tonClickTimer(PT:=tDoubleClickTime);
tonHoldTimer(PT:=tHoldTime);
cClickCnt(CU:=bButton, PV:=2);

// 点击检测
IF bButton AND cClickCnt.CV=1 THEN
	nStep := 1;												// 检测到单击
ELSIF bButton AND cClickCnt.CV=2 THEN
	nStep := 2;												// 检测到双击，进入双击+HOLD模式检测
END_IF



IF tonClickTimer.Q AND NOT bButton THEN						// 第一次单击后开启tonClickTimer计时器，计时器触发且没有检测到按钮按下，则将按键计数器复位，并将状态nstep=0，恢复到默认无按键按下状态。
	cClickCnt(RESET:= TRUE);
	nStep	:= 0;
ELSIF tonClickTimer.Q AND bButton AND cClickCnt.CV=1 THEN	// 第一次单击后开启tonClickTimer计时器，计时器触发且检测到按钮一直被按下。
	nStep := 3;												// 进入单击+HOLD模式
END_IF

// 按键计数器自复位
IF cClickCnt.Q THEN
	cClickCnt(reset:=TRUE);
END_IF




CASE nStep OF
	// 无按键状态，所有定时器计数器复位，两个输出变量bDoubleClickAndHold、bOnceClickAndHold置false
	0:
		tonClickTimer(IN := FALSE);
		tonHoldTimer(IN:=FALSE);
		cClickCnt(RESET:= FALSE);
		bDoubleClickAndHold := FALSE;
		bOnceClickAndHold:=FALSE;
	
	//点击模式检测
	1:
		tonClickTimer(IN:=TRUE);
		
	// 双击+hold检测
	2:
		tonHoldTimer(IN:=TRUE);								//开启hold时间计时器
		
		IF tonHoldTimer.Q AND bButton THEN					// 如果Hold时间满足，即为双击+hold状态
			bDoubleClickAndHold := TRUE;
		END_IF
		
		IF NOT bButton THEN									// 检测到按键释放，所有计时器计数器、输出状态复位
			bDoubleClickAndHold := FALSE;
			tonClickTimer(IN:=FALSE);
			tonHoldTimer(IN:=FALSE);
			cClickCnt(RESET:= TRUE);
			nStep:=0;
		END_IF
	
	// 单击+HOLD模式	
	3:
		IF tonClickTimer.Q AND bButton THEN					// 单击的hold时根据tonClickTimer时间来测量的，时间满足且按键未松，则为单击+hold
			bOnceClickAndHold := TRUE;
		END_IF
		
		IF NOT bButton THEN									// 检测到按键释放，所有计时器计数器、输出状态复位
			bOnceClickAndHold := FALSE;
			tonClickTimer(IN:=FALSE);
			cClickCnt(RESET:= TRUE);
			nStep:=0;
		END_IF
		
END_CASE

END_FUNCTION_BLOCK

// ---- POUs/TBoxCtrl.TcPOU
PROGRAM TBoxCtrl
VAR
END_VAR

IF bPumpMotor_Enable_TBox OR bPumpMotor_Enable_UpperUI THEN
	bPumpMotor_Enable:=TRUE;
ELSE
	bPumpMotor_Enable:=FALSE;
END_IF
	
IF bLeftArm_SV1_TBox OR bLeftArm_SV1_UpperUI THEN
	bLeftArm_SV1:=TRUE;
ELSE
	bLeftArm_SV1:=FALSE;
END_IF

IF bLeftArm_SV2_TBox OR bLeftArm_SV2_UpperUI THEN
	bLeftArm_SV2:=TRUE;
ELSE
	bLeftArm_SV2:=FALSE;
END_IF

IF bLeftArm_SV3_TBox OR bLeftArm_SV3_UpperUI THEN
	bLeftArm_SV3:=TRUE;
ELSE
	bLeftArm_SV3:=FALSE;
END_IF

IF bLeftArm_SV4_TBox OR bLeftArm_SV4_UpperUI THEN
	bLeftArm_SV4:=TRUE;
ELSE
	bLeftArm_SV4:=FALSE;
END_IF

IF bLeftArm_SV5_TBox OR bLeftArm_SV5_UpperUI THEN
	bLeftArm_SV5:=TRUE;
ELSE
	bLeftArm_SV5:=FALSE;
END_IF

IF bLeftArm_SV6_TBox OR bLeftArm_SV6_UpperUI THEN
	bLeftArm_SV6:=TRUE;
ELSE
	bLeftArm_SV6:=FALSE;
END_IF

IF bLeftArm_SV7_TBox OR bLeftArm_SV7_UpperUI THEN
	bLeftArm_SV7:=TRUE;
ELSE
	bLeftArm_SV7:=FALSE;
END_IF

IF bLeftArm_SV8_TBox OR bLeftArm_SV8_UpperUI THEN
	bLeftArm_SV8:=TRUE;
ELSE
	bLeftArm_SV8:=FALSE;
END_IF




IF bRightArm_SV1_TBox OR bRightArm_SV1_UpperUI THEN
	bRightArm_SV1:=TRUE;
ELSE
	bRightArm_SV1:=FALSE;
END_IF

IF bRightArm_SV2_TBox OR bRightArm_SV2_UpperUI THEN
	bRightArm_SV2:=TRUE;
ELSE
	bRightArm_SV2:=FALSE;
END_IF

IF bRightArm_SV3_TBox OR bRightArm_SV3_UpperUI THEN
	bRightArm_SV3:=TRUE;
ELSE
	bRightArm_SV3:=FALSE;
END_IF

IF bRightArm_SV4_TBox OR bRightArm_SV4_UpperUI THEN
	bRightArm_SV4:=TRUE;
ELSE
	bRightArm_SV4:=FALSE;
END_IF

IF bRightArm_SV5_TBox OR bRightArm_SV5_UpperUI THEN
	bRightArm_SV5:=TRUE;
ELSE
	bRightArm_SV5:=FALSE;
END_IF

IF bRightArm_SV6_TBox OR bRightArm_SV6_UpperUI THEN
	bRightArm_SV6:=TRUE;
ELSE
	bRightArm_SV6:=FALSE;
END_IF

IF bRightArm_SV7_TBox OR bRightArm_SV7_UpperUI THEN
	bRightArm_SV7:=TRUE;
ELSE
	bRightArm_SV7:=FALSE;
END_IF

IF bRightArm_SV8_TBox OR bRightArm_SV8_UpperUI THEN
	bRightArm_SV8:=TRUE;
ELSE
	bRightArm_SV8:=FALSE;
END_IF

END_PROGRAM

// ---- POUs/AxisStatus.TcPOU
PROGRAM AxisStatus
VAR
	


RE:AxisStatusReadErrorCode;





END_VAR

axis_RightArm_Left();
axis_RightArm_Right();
axis_RightArm_Wrist();
axis_RightArm_Lift();
axis_LeftArm_Left();
axis_LeftArm_Right();
axis_LeftArm_Wrist();
axis_LeftArm_Lift();
axis_SmallGate_Left();
axis_SmallGate_Right();
axis_BigGate_Left();
axis_BigGate_Right();
axis_BackGate_Left();
axis_BackGate_Right();

END_PROGRAM

// ---- POUs/AxisStatusReadErrorCode.TcPOU
FUNCTION_BLOCK AxisStatusReadErrorCode
VAR_INPUT
	AxisName				:AXIS_REF;

END_VAR
VAR_OUTPUT
	ErrorCode				:STRING;
	nMainAlarmCode			: USINT;
	nSubAlarmCode			: USINT;
END_VAR
VAR
	fbReadDriverSDO			: FB_EcCoeSdoRead;
	receivedAlarmCode		: UDINT;
//	nMainAlarmCode			: USINT;
//	nSubAlarmCode			: USINT;
	
	
END_VAR

fbReadDriverSDO(
	sNetId:= '192.168.1.20.1.1', 
	nSlaveAddr:= 1014, 
	nSubIndex:= 16#02, 
	nIndex:= 16#4DA0, 
	pDstBuf:= ADR(receivedAlarmCode), 
	cbBufLen:= 8, 
	bExecute:= , 
	tTimeout:= , 
	bBusy=> , 
	bError=> , 
	nErrId=> , 
	cbRead=> );
	
//0111 1111 1111 1111
//7F		FF
//nMainAlarmCode  := receivedAlarmCode AND SHL(16#0000007F, 8);
//nSubAlarmCode	:= receivedAlarmCode AND SHL(16#000000FF, 0);
nMainAlarmCode := TO_USINT(SHR(receivedAlarmCode, 8)) AND (16#7F);
nSubAlarmCode := TO_USINT(receivedAlarmCode) AND (16#FF);

END_FUNCTION_BLOCK

// ---- POUs/LedControl.TcPOU
PROGRAM LedControl
VAR
	
	
	
	
END_VAR

END_PROGRAM

// ---- POUs/LedLogic.TcPOU
FUNCTION_BLOCK LedLogic
VAR_INPUT
END_VAR
VAR_OUTPUT
END_VAR
VAR
END_VAR

END_FUNCTION_BLOCK

// ---- POUs/ArmFK_bak.TcPOU
FUNCTION ArmFK_bak : Points
VAR_INPUT
	theta1:LREAL;
	theta2:LREAL;
END_VAR
VAR
	// 中间变量
	theta1_rad:LREAL;
	theta2_rad:LREAL;
	rr:LREAL;						//r变量被倍福占用了，所以此处用rr
	u:LREAL;
	angle_ACD:LREAL;
	angle_DCE:LREAL;
	angle_ACF:LREAL;
	angle_FCG:LREAL;
	angle_FCI:LREAL;
	
	// 输出
	points : Points;

END_VAR

(*

theta1_rad := DEG_TO_RAD(theta1);
theta2_rad := DEG_TO_RAD(theta2);


rr := SQRT(EXPT((2*w+f*COS(theta1_rad)-g*COS(theta2_rad)),2) + EXPT((f*SIN(theta1_rad)-g*SIN(theta2_rad)),2));  

u := SQRT(EXPT((2*w-g*COS(theta2_rad)),2) + EXPT((-g*SIN(theta2_rad)),2));


angle_ACD := ACOS((rr*rr+f*f-u*u)/(2*rr*f));


angle_DCE := ACOS((rr*rr + i*i -h*h)/(2*rr*i));


angle_ACF := angle_ACD + angle_DCE + DEG_TO_RAD(angle_FCE);


angle_FCG := angle_ACF - theta1_rad;


angle_FCI := PI - angle_FCG;
points.x := w + f*COS(theta1_rad) + n*COS(angle_FCI);
points.y := f*SIN(theta1_rad) + n*SIN(angle_FCI);

ArmLeftFK := points;

*)

END_FUNCTION

// ---- POUs/ArmIK_bak.TcPOU
FUNCTION ArmIK_bak : Angles
VAR_INPUT
	x:LREAL;
	y:LREAL;
END_VAR
VAR
	
	// 中间量
	p:LREAL;
	q:LREAL;
	l:LREAL;
	k:LREAL;
	angle_CAF:LREAL;	
	angle_OAF:LREAL;
	theta1:LREAL;
	theta2:LREAL;
	angle_ACF:LREAL;
	angle_ACE:LREAL;
	angle_CAE:LREAL;
	angle_EAB:LREAL;
	angle_EBA:LREAL;
	angle_DBE:LREAL;
	
	// 输出
	angles		:Angles;
	
END_VAR

// TWINCAT 角度换算以弧度为单位
(*

p := SQRT((x-w)*(x-w)+y*y);
q := SQRT(x*x + y*y);
 
//n := SQRT(i*i+j*j-2*i*j*COS(DEG_TO_RAD(angle_a)));
angle_CAF := ACOS((f*f+p*p-n*n)/(2*f*p));
angle_OAF := ACOS((w*w+p*p-q*q)/(2*w*p));
theta1 := PI-angle_CAF-angle_OAF;

angle_ACF := ACOS((f*f+n*n-p*p)/(2*f*n));
//angle_FCE := ACOS((n*n+i*i-j*j)/(2*n*i));
angle_ACE := angle_ACF - DEG_TO_RAD(angle_FCE);
l := SQRT(i*i+f*f-2*i*f*COS(angle_ACE));
angle_CAE := ACOS((f*f+l*l-i*i)/(2*f*l));
angle_EAB := PI-theta1 - angle_CAE;
k := SQRT(l*l + 4*w*w - 4*l*w*COS(angle_EAB));
angle_EBA := ACOS((k*k+4*w*w-l*l)/(4*k*w));
angle_DBE := ACOS((g*g+k*k-h*h)/(2*g*k));
theta2 := angle_EBA + angle_DBE;

angles.theta1_right := RAD_TO_DEG(theta1);
angles.theta2_left := RAD_TO_DEG(theta2);


ArmLeftIK := angles;

*)

END_FUNCTION

// ---- POUs/ArmMove.TcPOU
PROGRAM ArmMove
VAR
	
	point												:Points;					// 当前腕关节坐标
	target_angle										:Angles;					// 臂左右电机目标角度
	manualState											:USINT;						// 手动控制状态标志位，0
	speed												:REAL := 1;					// 笛卡尔坐标位移速度
	x													:REAL;						// 腕关节目标位置x
	y													:REAL;						// 腕关节目标位置y
	wrist_angle											:REAL;
	wrist_MoveAbs										:MC_MoveAbsolute;
	
	LeftArm_Right_ExtPosGen_Enable						:MC_ExtSetPointGenEnable;
	LeftArm_Right_ExtPosGen_Disable                     :MC_ExtSetPointGenDisable;
	LeftArm_Left_ExtPosGen_Enable                       :MC_ExtSetPointGenEnable;
	LeftArm_Left_ExtPosGen_Disable	                    :MC_ExtSetPointGenDisable;
	
	fb_SerialCom		:FB_SerialCom;					//串口
	wrist_angle_int		:INT;
	wrist_angle_byte	:BYTE;
	
	
END_VAR

axis_LeftArm_Left();
axis_LeftArm_Right();
ExtPosGen();

// 外部位置发生器失能
LeftArm_Right_ExtPosGen_Enable.Execute 		:= FALSE;
LeftArm_Right_ExtPosGen_Disable.Execute 	:= FALSE;
LeftArm_Left_ExtPosGen_Enable.Execute 		:= FALSE;
LeftArm_Left_ExtPosGen_Disable.Execute 		:= FALSE;

IF bManualCtrl_Part_LeftArm_Left THEN
	
	// 运动学正解出当前腕关节点坐标
	point := ArmFK(axis_LeftArm_Right.NcToPlc.ActPos, axis_LeftArm_Left.NcToPlc.ActPos);
	
	// 用舵机进行程序验证的串口背景通讯
	//BackgroundSerialCtrl();
	
	IF bAutoCtrl_Part_LeftWrist THEN
		
		wrist_angle := WristIK(point.x, point.y);		// 逆解出腕电机角度
		wrist_angle_int:= TO_INT(wrist_angle);
		
		// 用舵机进行程序验证的串口测试
		//wrist_angle_byte:= INT_TO_BYTE(wrist_angle_int);
		//fb_SerialCom(TxBuffer:= TxBuffer, RxBuffer:= RxBuffer, angle:= wrist_angle_byte);	
		
		wrist_MoveAbs(Axis:= axis_LeftArm_Wrist, Execute:= TRUE, Position:= wrist_angle, Velocity:= 5, Acceleration:= 10, Deceleration:= , Jerk:= , BufferMode:= , 
					  Options:= , Done=> , Busy=> , Active=> , CommandAborted=> , Error=> , ErrorID=> );		// 腕电机走绝对定位
	END_IF
	

	IF bLeftArm_Forward THEN
		x := point.x;
		y := point.y + speed;
		target_angle := ArmIK(x, y);
		manualState := 1;
		
	ELSIF bLeftArm_Backward THEN
	
		x := point.x;
		y := point.y - speed;
		target_angle := ArmIK(x, y);
		manualState := 1;
		
	ELSIF bLeftArm_Left THEN
		
		x := point.x - speed;
		y := point.y;
		target_angle := ArmIK(x, y);
		manualState := 1;
		
	ELSIF bLeftArm_Right THEN
		
		x := point.x + speed;
		y := point.y;
		target_angle := ArmIK(x, y);
		manualState := 1;
		
	ELSE
		manualState := 0;
	END_IF
	
	
	
	CASE manualState OF
		0:
			LeftArm_Right_ExtPosGen_Enable.Execute 		:= FALSE;
			LeftArm_Right_ExtPosGen_Disable.Execute 	:= TRUE;
			LeftArm_Left_ExtPosGen_Enable.Execute 		:= FALSE;
			LeftArm_Left_ExtPosGen_Disable.Execute 		:= TRUE;
		
		1:
			LeftArm_Right_ExtPosGen_Enable.Execute := TRUE;
			LeftArm_Left_ExtPosGen_Enable.Execute := TRUE;
			IF axis_LeftArm_Right.Status.ExtSetPointGenEnabled AND axis_LeftArm_Left.Status.ExtSetPointGenEnabled THEN
				MC_ExtSetPointGenFeed(
					Position:= target_angle.theta1_right, 
					Velocity:= 30,  
					Acceleration:= 10,  
					Direction:= 1, 
					Axis:= axis_LeftArm_Right);
		
				MC_ExtSetPointGenFeed(
					Position:= target_angle.theta2_left, 
					Velocity:= 30,  
					Acceleration:= 10,  
					Direction:= 1, 
					Axis:= axis_LeftArm_Left);
			END_IF
	END_CASE

//ELSE

END_IF

ACTION ExtPosGen:
LeftArm_Right_ExtPosGen_Enable(
	Axis:= axis_LeftArm_Right, 
	Execute:= LeftArm_Right_ExtPosGen_Enable.Execute, 
	Position:= , 
	PositionType:= , 
	Done=> , 
	Busy=> , 
	Error=> , 
	ErrorID=> , 
	Enabled=> );
	
LeftArm_Right_ExtPosGen_Disable(
	Axis:= axis_LeftArm_Right, 
	Execute:= LeftArm_Right_ExtPosGen_Disable.Execute, 
	Done=> , 
	Busy=> , 
	Error=> , 
	ErrorID=> , 
	Enabled=> );
	
LeftArm_Left_ExtPosGen_Enable(
	Axis:= axis_LeftArm_Left, 
	Execute:= LeftArm_Left_ExtPosGen_Enable.Execute, 
	Position:= , 
	PositionType:= , 
	Done=> , 
	Busy=> , 
	Error=> , 
	ErrorID=> , 
	Enabled=> );
	
LeftArm_Left_ExtPosGen_Disable(
	Axis:= axis_LeftArm_Left, 
	Execute:= LeftArm_Left_ExtPosGen_Disable.Execute, 
	Done=> , 
	Busy=> , 
	Error=> , 
	ErrorID=> , 
	Enabled=> );
END_ACTION

END_PROGRAM

// ---- POUs/AxisCaliHomePos.TcPOU
PROGRAM AxisCaliHomePos
VAR
	writeParam		:MC_WriteParameter;
	bWriteParam_DO	:BOOL;
	
END_VAR


writeParam(
	Axis:= axis_RightArm_Wrist, 
	Execute:= bWriteParam_DO, 
	ParameterNumber:= AxisEncoderOffset, 
	Value:= -2, 
	Done=> , 
	Busy=> , 
	Error=> , 
	ErrorID=> );

END_PROGRAM

// ---- POUs/Gate_Back_Move.TcPOU
PROGRAM Gate_Back_Move
VAR
	
	backGateGearIn					:MC_GearIn;
	backGateGearOut					:MC_GearOut;	                    			
	backGateLeftAxisJog 			:MC_Jog;
	backGateLeftAxisMoveAbs			:MC_MoveAbsolute;		// 后龙门MoveAbs(实际上电子齿轮的Master轴axis_BackGate_Left的Mc_MoveAbsolute)                    			
	
	//bBackGate_Gearin_do				:BOOL:=TRUE;

	nBackGate_Speed					:LREAL:=5;		// 后龙门移动速度
	nBackGate_MoveAbs_TarPos		:LREAL;			// 后龙门MoveAbs目标位置	
	
	
END_VAR

// Mc_Jog
backGateLeftAxisJog(
	Axis:= axis_BackGate_Left, 
	JogForward:= bBackGate_Down AND bManualCtrl_Asm_BackGate, 
	JogBackwards:= bBackGate_Up AND bManualCtrl_Asm_BackGate, 
	Mode:= MC_JOGMODE_CONTINOUS, 
	Position:= , 
	Velocity:= nBackGate_Speed, 
	Acceleration:= , 
	Deceleration:= , 
	Jerk:= , 
	Done=> , 
	Busy=> , 
	Active=> , 
	CommandAborted=> , 
	Error=> , 
	ErrorID=> );

// Mc_MoveAbs
backGateLeftAxisMoveAbs(
	Axis:= axis_BackGate_Left, 
	Execute:= bBackGate_MoveAbs AND bManualCtrl_Asm_BackGate, 
	Position:= (-1)*nBackGate_MoveAbs_TarPos, 						// 反转升，所以绝对位置也要反着
	Velocity:= nBackGate_Speed, 
	Acceleration:= , 
	Deceleration:= , 
	Jerk:= , 
	BufferMode:= , 
	Options:= , 
	Done=> , 
	Busy=> , 
	Active=> , 
	CommandAborted=> , 
	Error=> , 
	ErrorID=> );	

	
backGateGearIn(
	Master:= axis_BackGate_Left, 
	Slave:= axis_BackGate_Right, 
	Execute:= bBackGate_GearIn_do, 
	RatioNumerator:= 1, 
	RatioDenominator:= 1, 
	Acceleration:= , 
	Deceleration:= , 
	Jerk:= , 
	BufferMode:= , 
	Options:= , 
	InGear=> , 
	Busy=> , 
	Active=> , 
	CommandAborted=> , 
	Error=> , 
	ErrorID=> );


backGateGearOut(
	Slave:= axis_BackGate_Right, 
	Execute:= NOT bBackGate_GearIn_do, 
	Options:= , 
	Done=> , 
	Busy=> , 
	Error=> , 
	ErrorID=> );

END_PROGRAM

// ---- POUs/Gate_Small_Move.TcPOU
PROGRAM Gate_Small_Move
VAR
	smallGateGearIn				:MC_GearIn;				// 小龙门电子齿轮，LeftAxis为Master
	smallGateGearOut			:MC_GearOut;			// 小龙门电子齿轮取消啮合
	smallGateLeftAxisJog		:MC_Jog;				// 小龙门左轴(电子齿轮的Master轴)MC_Jog
	smallGateLeftAxisMoveAbs	:MC_MoveAbsolute;		// 小龙门MoveAbs(实际上电子齿轮的Master轴axis_SmallGate_Left的Mc_MoveAbsolute)
	
	// 默认为啮合状态，当激活大龙门左轴或者右轴的手动控制时bManualCtrl_Part_SmallGate_Left为true
	//或bManualCtrl_Part_SmallGate_Right为True，会把此变量置false
	//bSmallGate_Gearin_do		:BOOL:=TRUE;
	
	nSmallGate_Speed					:LREAL:=2;		// 小龙门移动速度
	nSmallGate_MoveAbs_TarPos			:LREAL;			// 小龙门MoveAbs目标位置
	
END_VAR

// SmallGate Mc_Jog
smallGateLeftAxisJog(
	Axis:= axis_SmallGate_Left, 
	JogForward:= bSmallGate_Down AND bManualCtrl_Asm_SmallGate, 
	JogBackwards:= bSmallGate_Up AND bManualCtrl_Asm_SmallGate, 
	Mode:= MC_JOGMODE_CONTINOUS, 
	Position:= , 
	Velocity:= nSmallGate_Speed, 
	Acceleration:= , 
	Deceleration:= , 
	Jerk:= , 
	Done=> , 
	Busy=> , 
	Active=> , 
	CommandAborted=> , 
	Error=> , 
	ErrorID=> );

// SmallGate Mc_MoveAbsolute
smallGateLeftAxisMoveAbs(
	Axis:= axis_SmallGate_Left, 
	Execute:= bSmallGate_MoveAbs AND bManualCtrl_Asm_SmallGate, 
	Position:= (-1)*nSmallGate_MoveAbs_TarPos, 						// 反转升，所以绝对位置也要反着
	Velocity:= nSmallGate_Speed, 
	Acceleration:= , 
	Deceleration:= , 
	Jerk:= , 
	BufferMode:= , 
	Options:= , 
	Done=> , 
	Busy=> , 
	Active=> , 
	CommandAborted=> , 
	Error=> , 
	ErrorID=> );
	
smallGateGearIn(
	Master:= axis_SmallGate_Left, 
	Slave:= axis_SmallGate_Right, 
	Execute:= bSmallGate_Gearin_do, 
	RatioNumerator:= -1, 
	RatioDenominator:= 1, 
	Acceleration:= , 
	Deceleration:= , 
	Jerk:= , 
	BufferMode:= , 
	Options:= , 
	InGear=> , 
	Busy=> , 
	Active=> , 
	CommandAborted=> , 
	Error=> , 
	ErrorID=> );
	
	
smallGateGearOut(
	Slave:= axis_SmallGate_Right, 
	Execute:= NOT bSmallGate_Gearin_do, 
	Options:= , 
	Done=> , 
	Busy=> , 
	Error=> , 
	ErrorID=> );

END_PROGRAM

// ---- POUs/Serial/BmsSerial.TcPOU
PROGRAM BmsSerial
VAR
	// 发送命令
	sendQueryBmsCmd 			:SendData;
	
	// 定时器5s触发一次
	timer1						:TON;
	timer1Trigger				:BOOL		:= TRUE;
	time5s						:TIME 		:=T#5S;

	
	// 接收命令
	recvDataFromBms				:ReceiveData;
	prefixRecvData				:ARRAY[1..2] OF BYTE		:=[16#DD,16#03];
	suffixRecvData				:BYTE						:=16#77;
	receivedData				:ARRAY[1..45] OF BYTE;
	bReceived					:BOOL;
	
	//test

	
	
END_VAR


//定时器
timer1(IN:= timer1Trigger, PT:= time5s, Q=> , ET=> );
IF timer1.Q THEN
	timer1Trigger:= FALSE;
	
	// 发送查询bms命令
	sendQueryBmsCmd(
		pSendData:= ADR(queryBmsStatusCmd), 
		Length:= queryBmsStatusCmdLen, 
		Busy=> , 
		Error=> , 
		TXbuffer:= TxBuffer);
		//sendQueryBmsCmd(SendString:='DDA50300FFFD77' , Busy=> , Error=> , TXbuffer:= TxBuffer);
		
		
	// 接收bms数据
	recvDataFromBms(
		pPrefix:= ADR(prefixRecvData), 
		LenPrefix:= 2, 
		pSuffix:= ADR(suffixRecvData), 
		LenSuffix:= 1, 
		pReceiveData:= ADR(receivedData), 
		SizeReceiveData:= SIZEOF(receivedData), 
		Timeout:= T#2S, 
		Reset:= , 
		DataReceived=> bReceived, 
		busy=> , 
		Error=> , 
		RxTimeout=> , 
		LenReceiveData=> , 
		RXbuffer:= RxBuffer);
	
		
		
		
	// 串口数据处理	
	Battery_TotalVoltage 		:=	( BYTE_TO_UINT(receivedData[5]) * 256 + BYTE_TO_UINT(receivedData[6]) ) * 10 * 0.001;				//voltage, receivedData[5][6]，Unit:V
	Battery_TotalCurrent 		:= UINT_TO_INT( BYTE_TO_UINT(receivedData[7]) * 256 + BYTE_TO_UINT(receivedData[8]) ) * 10 * 0.001;		//current, receivedData[7][8]，Unit:A, minus:discharging, plus:charging
	Battery_RemainCapacity		:= ( BYTE_TO_UINT(receivedData[9]) * 256 + BYTE_TO_UINT(receivedData[10]) ) * 10 * 0.001;				//remain capacity, receivedData[9][10], Unit:Ah	
	Battery_NominalCapacity		:= ( BYTE_TO_UINT(receivedData[11]) * 256 + BYTE_TO_UINT(receivedData[12]) ) * 10 * 0.001;				//nominal capacity, receivedData[9][10], Unit:Ah	
	Battery_CycleNum			:= BYTE_TO_UINT(receivedData[13]) * 256 + BYTE_TO_UINT(receivedData[14]) ;								//cycle num, received[13][14], Unit: number of times
	Battery_ProtectionMode		:= SHL(TO_WORD(receivedData[21]),8) OR TO_WORD(receivedData[22]);										//protection word, received[21][22], protection word list is in Robot_Status_Info
	Battery_RSOC	     		:= BYTE_TO_USINT(receivedData[24]);																		//remain soc, receivedData[24], Unit:%
	Battery_FETStatus			:= receivedData[25];																					//fet status word
	Battery_humidity			:= BYTE_TO_USINT(receivedData[34]);																		//humidity, unit:%
	Battery_WarningStatus		:= SHL(TO_WORD(receivedData[35]),8) OR TO_WORD(receivedData[36]);										//warning status word, received[35][36], warning status word list is in Robot_Status_Info
	
	// 电池充放电状态判断
	IF Battery_TotalCurrent > 0 THEN
		bBattery_Charging 		:= TRUE;
		bBattery_DisCharging	:= FALSE;
	ELSIF Battery_TotalCurrent <0 THEN
		bBattery_Charging := FALSE;
		bBattery_DisCharging := TRUE;
	ELSE
		bBattery_Charging 		:= FALSE;
		bBattery_DisCharging	:= FALSE;
	END_IF
	
	// 电池剩余百分比计算
	IF Battery_NominalCapacity <> 0 THEN
		lrBattery_RemainCapacity_Pecent		:=	(Battery_RemainCapacity/Battery_NominalCapacity)*100;	
	END_IF

	
	// Battery_ProtectionMode，电池保护标志位状态处理
	bSingleCellOvervoltageProtection     := (Battery_ProtectionMode AND 16#0001) <> 0;			// bit0: 单体过压保护    
	bSingleCellUndervoltageProtection    := (Battery_ProtectionMode AND 16#0002) <> 0;			// bit1: 单体欠压保护    
	bWholeGroupOvervoltageProtection     := (Battery_ProtectionMode AND 16#0004) <> 0;			// bit2: 整组过压保护    
	bWholeGroupUndervoltageProtection    := (Battery_ProtectionMode AND 16#0008) <> 0;			// bit3: 整组欠压保护    
	bChargingOverTemperatureProtection   := (Battery_ProtectionMode AND 16#0010) <> 0;			// bit4: 充电过温保护    
	bChargingLowTemperatureProtection    := (Battery_ProtectionMode AND 16#0020) <> 0;			// bit5: 充电低温保护    
	bDischargingOverTemperatureProtection:= (Battery_ProtectionMode AND 16#0040) <> 0;			// bit6: 放电过温保护    
	bDischargingLowTemperatureProtection := (Battery_ProtectionMode AND 16#0080) <> 0;			// bit7: 放电低温保护    
	bChargingOvercurrentProtection       := (Battery_ProtectionMode AND 16#0100) <> 0;			// bit8: 充电过流保护    
	bDischargingOvercurrentProtection    := (Battery_ProtectionMode AND 16#0200) <> 0;			// bit9: 放电过流保护    
	bShortCircuitProtection              := (Battery_ProtectionMode AND 16#0400) <> 0;			// bit10: 短路保护     
	bFrontEndDetectionICError            := (Battery_ProtectionMode AND 16#0800) <> 0;			// bit11: 前端检测IC错误 
	bSoftwareLockedMOS                   := (Battery_ProtectionMode AND 16#1000) <> 0;			// bit12: 软件锁定MOS  
	bChargingMOSBreakdownFlag            := (Battery_ProtectionMode AND 16#2000) <> 0;			// bit13: 充电MOS击穿标志
	bDischargingMOSBreakdownFlag         := (Battery_ProtectionMode AND 16#4000) <> 0;			// bit14: 放电MOS击穿标志
		
	// Battery_FETStatus, 电池MOSFET状态标志位处理
	bChargeMOSStatus    				 := (Battery_FETStatus AND 16#01) <> 0; 					// bit0: 充电MOS状态
	bDischargeMOSStatus 				 := (Battery_FETStatus AND 16#02) <> 0; 					// bit1: 放电MOS状态
	bCurrentLimitStatus 				 := (Battery_FETStatus AND 16#04) <> 0; 					// bit2: 限流模块状态 
	bHeatingStatus      				 := (Battery_FETStatus AND 16#08) <> 0; 					// bit3: 加热模块状态 
	
	//Battery_WarningStatus, 电池报警状态处理
	bSingleCellHighVoltageWarning     	 := (Battery_WarningStatus AND 16#0001) <> 0; 			// bit0: 单体高压告警  
	bSingleCellLowVoltageWarning      	 := (Battery_WarningStatus AND 16#0002) <> 0; 			// bit1: 单体低压告警  
	bWholeGroupHighVoltageWarning     	 := (Battery_WarningStatus AND 16#0004) <> 0; 			// bit2: 整组高压告警  
	bWholeGroupLowVoltageWarning      	 := (Battery_WarningStatus AND 16#0008) <> 0; 			// bit3: 整组低压告警  
	bChargingHighTemperatureWarning   	 := (Battery_WarningStatus AND 16#0010) <> 0; 			// bit4: 充电高温告警  
	bChargingLowTemperatureWarning    	 := (Battery_WarningStatus AND 16#0020) <> 0; 			// bit5: 充电低温告警  
	bDischargingHighTemperatureWarning	 := (Battery_WarningStatus AND 16#0040) <> 0; 			// bit6: 放电高温告警  
	bDischargingLowTemperatureWarning 	 := (Battery_WarningStatus AND 16#0080) <> 0; 			// bit7: 放电低温保护  
	bChargingHighCurrentWarning       	 := (Battery_WarningStatus AND 16#0100) <> 0; 			// bit8: 充电电流大告警 
	bDischargingHighCurrentWarning    	 := (Battery_WarningStatus AND 16#0200) <> 0; 			// bit9: 放电电流大告警 
	bSingleCellVoltageDifferenceWarning  := (Battery_WarningStatus AND 16#0400) <> 0; 			// bit10: 单体压差大告警
	bLowCapacityWarning               	 := (Battery_WarningStatus AND 16#0800) <> 0; 			// bit11: 容量低告警  
	bReserved12                       	 := (Battery_WarningStatus AND 16#1000) <> 0; 			// bit12: 预留     
	bReserved13                       	 := (Battery_WarningStatus AND 16#2000) <> 0; 			// bit13: 预留     
	bReserved14                       	 := (Battery_WarningStatus AND 16#4000) <> 0; 			// bit14: 预留     
	
ELSE
	timer1Trigger:= TRUE;
END_IF

END_PROGRAM

// ---- POUs/Serial/BmsSerialBackground.TcPOU
PROGRAM BmsSerialBackground
VAR
	
END_VAR

BMSSerialCtrl(
	Mode:= SERIALLINEMODE_PC_COM_PORT, 
	pComIn:= ADR(pComIn), 
	pComOut:= ADR(pComOut), 
	SizeComIn:= SIZEOF(pComIN), 
	Error=> , 
	ErrorID=> , 
	TxBuffer:= TxBuffer, 
	RxBuffer:= RxBuffer);

END_PROGRAM
